{attribute 'pack_mode' := '1'}
TYPE ST_StartPathDataIn :
STRUCT
	iPath						: UINT;			// MM path ID (1-65536)
END_STRUCT
END_TYPE

(* stored: Version 1.1.0.1, ProductVersion 3.1.4024.5
   DUT ST_StartPathDataIn: Id {656e79c1-214c-408a-8ee3-d26e04b4fcac} *)
